ABB RAPID module: TCP_toolTest1.mod

MODULE TCP_toolTest1
	! Points are read in order of declaration.
  ! Please do not change the order of points!

  LOCAL PERS robtarget pTCP_Point1:=[[398.6034,-841.8726,356.7087],[0.439348459243774,-0.727854251861572,0.0786844119429588,-0.520586133003235],[-1,0,-4,0],[9E+09,9E+09,9E+09,9E+09,9E+09,9E+09]];
	LOCAL PERS robtarget pTCP_Point2:=[[538.3836,-778.2805,371.7353],[0.544624805450439,-0.177098587155342,-0.775396227836609,0.266046315431595],[-1,-1,-4,0],[9E+09,9E+09,9E+09,9E+09,9E+09,9E+09]];
	LOCAL PERS robtarget pTCP_Point3:=[[469.317,-708.0986,357.5158],[0.236785545945168,0.102643474936485,-0.746701538562775,0.613052845001221],[-1,-2,-4,0],[9E+09,9E+09,9E+09,9E+09,9E+09,9E+09]];
	LOCAL PERS robtarget pTCP_Point4:=[[432.8631,-786.813,401.7622],[7.84076200943673E-06,-0.381953865289688,-0.924181401729584,-4.92979097543866E-06],[-1,-1,-1,0],[9E+09,9E+09,9E+09,9E+09,9E+09,9E+09]];

ENDMODULE
